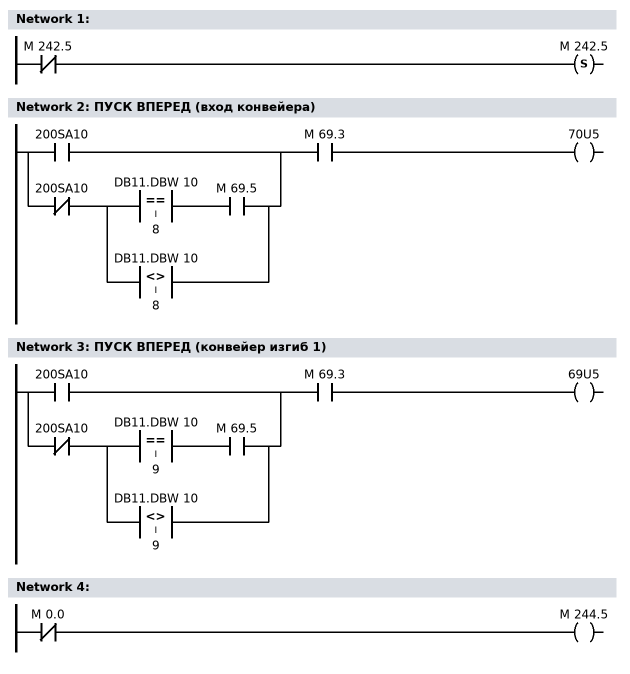
NETWORK
TITLE =
      AN    M 242.5;
      S     M 242.5;
NETWORK
TITLE = ПУСК ВПЕРЕД (вход конвейера)
      A(;
      O     "200SA10";
      O;
      AN    "200SA10";
      A(;
      A(;
      L     DB11.DBW 10;
      L     8;
      ==I;
      );
      A     M 69.5;
      O(;
      L     DB11.DBW 10;
      L     8;
      <>I;
      );
      );
      );
      A     M 69.3;
      =     "70U5";
NETWORK
TITLE = ПУСК ВПЕРЕД (конвейер изгиб 1)
      A(;
      O     "200SA10";
      O;
      AN    "200SA10";
      A(;
      A(;
      L     DB11.DBW 10;
      L     9;
      ==I;
      );
      A     M 69.5;
      O(;
      L     DB11.DBW 10;
      L     9;
      <>I;
      );
      );
      );
      A     M 69.3;
      =     "69U5";
NETWORK
TITLE =
      AN    M 0.0;
      =     M 244.5;
END_FUNCTION

FUNCTION FC 100 : VOID
VERSION : 0.1
BEGIN
// (block stored without names or comments; labels and parameter names are numbered)
NETWORK
TITLE =
      A     M 255.1;
      O(;
      A     DB11.DBX 1.6;
      A(;
      L     DB11.DBW 8;
      L     DB11.DBW 4;
      ==I;
      );
      );
      JCN   M001;
      AN    M 255.0;
      JCN   M001;
      L     DB11.DBW 4;
      L     100;
      +I;
      T     LW 100;
      L     101;
      <I;
      JC    M001;
      L     LW 100;
      L     104;
      >I;
      JC    M001;
      L     LW 100;
      OPN   DB [LW 100];
      CALL  "BLKMOV" (
           SRCBLK                   := P#DBX 0.0 BYTE 210,
           RET_VAL                  := LW 50,
           DSTBLK                   := P#DB99.DBX 0.0 BYTE 210);
M001: NOP   0;
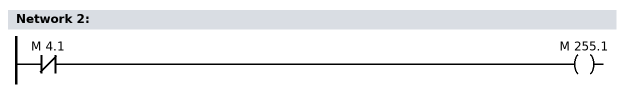
NETWORK
TITLE =
      AN    M 4.1;
      =     M 255.1;
NETWORK
TITLE =
      AN    DB11.DBX 2.0;
      JC    M002;
      L     DB11.DBW 8;
      L     100;
      +I;
      T     LW 100;
      L     101;
      <I;
      JC    M002;
      L     LW 100;
      L     104;
      >I;
      JC    M002;
      L     LW 100;
      OPN   DB [LW 100];
      CALL  "BLKMOV" (
           SRCBLK                   := P#DBX 0.0 BYTE 210,
           RET_VAL                  := LW 50,
           DSTBLK                   := P#DB100.DBX 0.0 BYTE 210);
      R     DB11.DBX 2.0;
M002: NOP   0;
NETWORK
TITLE =
      AN    DB11.DBX 1.6;
      JC    M003;
      L     DB11.DBW 8;
      L     100;
      +I;
      T     LW 100;
      L     101;
      <I;
      JC    M003;
      L     LW 100;
      L     104;
      >I;
      JC    M003;
      L     LW 100;
      OPN   DI [LW 100];
      CALL  "BLKMOV" (
           SRCBLK                   := P#DB100.DBX 0.0 BYTE 210,
           RET_VAL                  := LW 50,
           DSTBLK                   := P#DIX 0.0 BYTE 210);
      AN    T 1;
      JC    M003;
      R     DB11.DBX 1.6;
M003: NOP   0;
      A     DB11.DBX 1.6;
      L     S5T#1S;
      SD    T 1;
END_FUNCTION

FUNCTION FC 101 : VOID
VERSION : 0.1
BEGIN
// (block stored without names or comments; labels and parameter names are numbered)
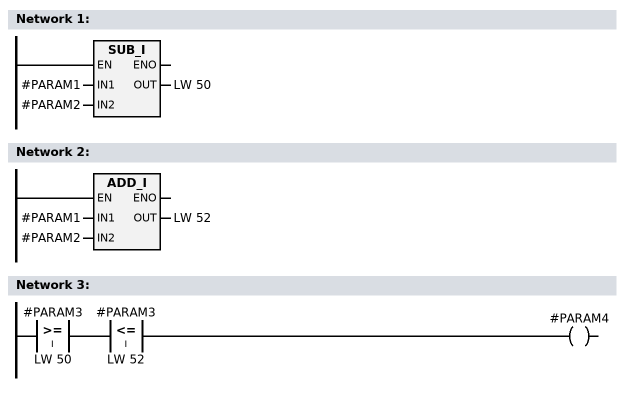
NETWORK
TITLE =
      L     #PARAM1;
      L     #PARAM2;
      -I;
      T     LW 50;
NETWORK
TITLE =
      L     #PARAM1;
      L     #PARAM2;
      +I;
      T     LW 52;
NETWORK
TITLE =
      A(;
      L     #PARAM3;
      L     LW 50;
      >=I;
      );
      A(;
      L     #PARAM3;
      L     LW 52;
      <=I;
      );
      =     #PARAM4;
END_FUNCTION

FUNCTION FC 102 : VOID
VERSION : 0.1
BEGIN
// (block stored without names or comments; labels and parameter names are numbered)
NETWORK
TITLE =
      L     DB12.DBW 516;
      L     256;
      >=I;
      JC    M001;
      L     DB12.DBW 516;
      L     2;
      *I;
      T     LD 0;
      L     LD 0;
      SLD   3;
      T     LD 0;
      L     DBW [LD 0];
      T     DB12.DBW 518;
      JU    M001;
      L     256;
      T     DB12.DBW 518;
M001: NOP   0;
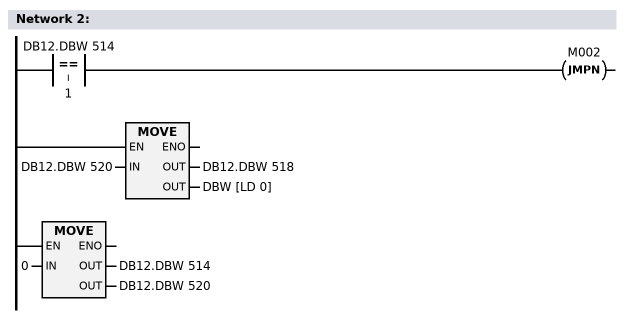
NETWORK
TITLE =
      L     DB12.DBW 514;
      L     1;
      ==I;
      JCN   M002;
      L     DB12.DBW 520;
      T     DB12.DBW 518;
      T     DBW [LD 0];
      L     0;
      T     DB12.DBW 514;
      T     DB12.DBW 520;
M002: NOP   0;
END_FUNCTION

FUNCTION FC 103 : VOID
VERSION : 0.1
BEGIN
// (block stored without names or comments; labels and parameter names are numbered)
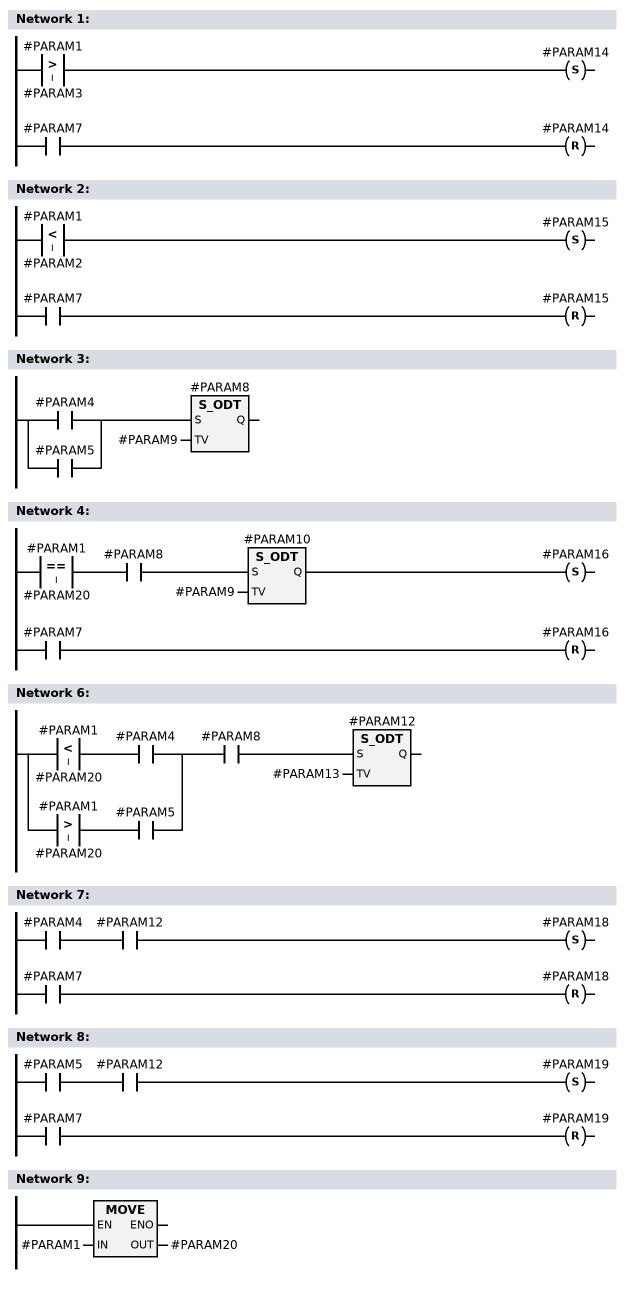
NETWORK
TITLE =
      A(;
      L     #PARAM1;
      L     #PARAM3;
      >I;
      );
      S     #PARAM14;
      A     #PARAM7;
      R     #PARAM14;
      NOP   0;
NETWORK
TITLE =
      A(;
      L     #PARAM1;
      L     #PARAM2;
      <I;
      );
      S     #PARAM15;
      A     #PARAM7;
      R     #PARAM15;
      NOP   0;
NETWORK
TITLE =
      A(;
      O     #PARAM4;
      O     #PARAM5;
      );
      L     #PARAM9;
      SD    #PARAM8;
      NOP   0;
      NOP   0;
      NOP   0;
      NOP   0;
NETWORK
TITLE =
      A(;
      A(;
      L     #PARAM1;
      L     #PARAM20;
      ==I;
      );
      A     #PARAM8;
      L     #PARAM9;
      SD    #PARAM10;
      NOP   0;
      NOP   0;
      NOP   0;
      A     #PARAM10;
      );
      S     #PARAM16;
      A     #PARAM7;
      R     #PARAM16;
      NOP   0;
NETWORK
TITLE =
      L     #PARAM20;
      L     #PARAM6;
      -I;
      T     LW 0;
      L     0;
      <I;
      JC    M001;
      JU    M002;
M001: L     0;
      T     LW 0;
M002: NOP   0;
      L     #PARAM20;
      L     #PARAM6;
      +I;
      T     LW 2;
      L     #PARAM1;
      L     LW 0;
      <I;
      JC    M003;
      L     #PARAM1;
      L     LW 2;
      >I;
      JC    M003;
      JU    M004;
M003: AN    #PARAM17;
      S     #PARAM17;
M004: R     #PARAM17;
NETWORK
TITLE =
      A(;
      A(;
      L     #PARAM1;
      L     #PARAM20;
      <I;
      );
      A     #PARAM4;
      O;
      A(;
      L     #PARAM1;
      L     #PARAM20;
      >I;
      );
      A     #PARAM5;
      );
      A     #PARAM8;
      L     #PARAM13;
      SD    #PARAM12;
      NOP   0;
      NOP   0;
      NOP   0;
      NOP   0;
NETWORK
TITLE =
      A     #PARAM4;
      A     #PARAM12;
      S     #PARAM18;
      A     #PARAM7;
      R     #PARAM18;
      NOP   0;
NETWORK
TITLE =
      A     #PARAM5;
      A     #PARAM12;
      S     #PARAM19;
      A     #PARAM7;
      R     #PARAM19;
      NOP   0;
NETWORK
TITLE =
      L     #PARAM1;
      T     #PARAM20;
END_FUNCTION

FUNCTION FC 104 : VOID
VERSION : 0.1
BEGIN
// (block stored without names or comments; labels and parameter names are numbered)
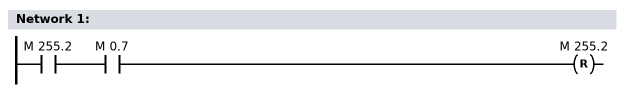
NETWORK
TITLE =
      A     M 255.2;
      A     M 0.7;
      R     M 255.2;
NETWORK
TITLE =
// (network holds code this reader does not know; not shown)
NETWORK
TITLE =
      L     MW 70;
      CAW;
      T     DB10.DBW 0;
      L     MW 72;
      CAW;
      T     DB10.DBW 2;
      L     MW 74;
      CAW;
      T     DB10.DBW 4;
      L     MW 76;
      CAW;
      T     DB10.DBW 6;
      L     MW 78;
      CAW;
      T     DB10.DBW 8;
      L     MW 80;
      CAW;
      T     DB10.DBW 10;
      L     MW 82;
      CAW;
      T     DB10.DBW 12;
      L     MW 84;
      CAW;
      T     DB10.DBW 14;
      L     MW 86;
      CAW;
      T     DB10.DBW 16;
      L     MW 88;
      CAW;
      T     DB10.DBW 18;
END_FUNCTION

FUNCTION FC 105 : VOID
VERSION : 0.1
BEGIN
// (block stored without names or comments; labels and parameter names are numbered)
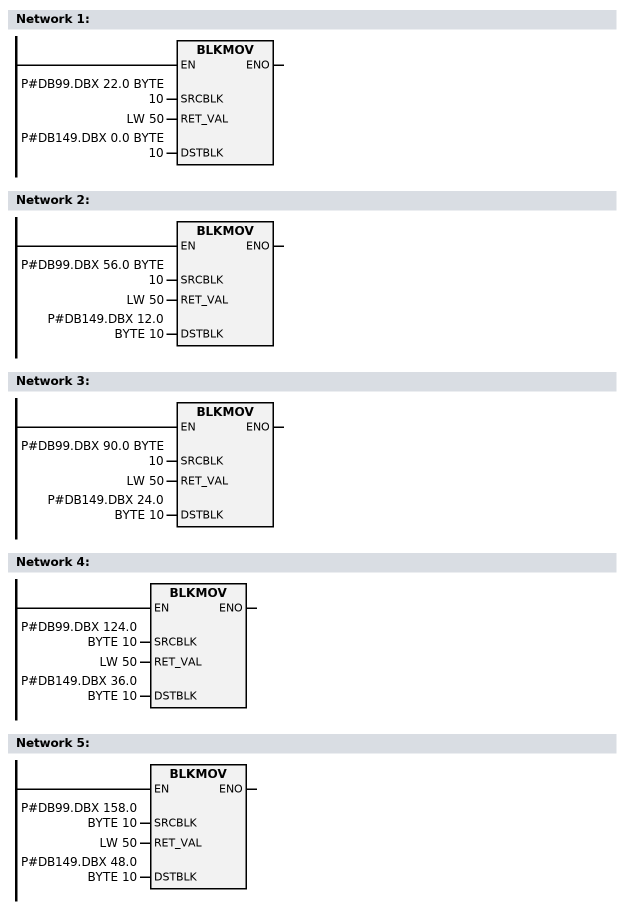
NETWORK
TITLE =
      CALL  "BLKMOV" (
           SRCBLK                   := P#DB99.DBX 22.0 BYTE 10,
           RET_VAL                  := LW 50,
           DSTBLK                   := P#DB149.DBX 0.0 BYTE 10);
NETWORK
TITLE =
      CALL  "BLKMOV" (
           SRCBLK                   := P#DB99.DBX 56.0 BYTE 10,
           RET_VAL                  := LW 50,
           DSTBLK                   := P#DB149.DBX 12.0 BYTE 10);
NETWORK
TITLE =
      CALL  "BLKMOV" (
           SRCBLK                   := P#DB99.DBX 90.0 BYTE 10,
           RET_VAL                  := LW 50,
           DSTBLK                   := P#DB149.DBX 24.0 BYTE 10);
NETWORK
TITLE =
      CALL  "BLKMOV" (
           SRCBLK                   := P#DB99.DBX 124.0 BYTE 10,
           RET_VAL                  := LW 50,
           DSTBLK                   := P#DB149.DBX 36.0 BYTE 10);
NETWORK
TITLE =
      CALL  "BLKMOV" (
           SRCBLK                   := P#DB99.DBX 158.0 BYTE 10,
           RET_VAL                  := LW 50,
           DSTBLK                   := P#DB149.DBX 48.0 BYTE 10);
END_FUNCTION

FUNCTION FC 110 : VOID
VERSION : 0.1
BEGIN
// (block stored without names or comments; labels and parameter names are numbered)
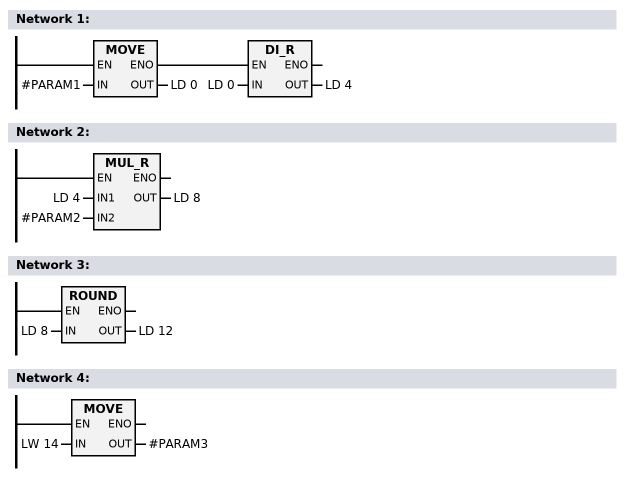
NETWORK
TITLE =
      A(;
      L     #PARAM1;
      T     LD 0;
      SET;
      SAVE;
      CLR;
      A     BR;
      );
      JNB   M001;
      L     LD 0;
      DTR;
      T     LD 4;
M001: NOP   0;
NETWORK
TITLE =
      L     LD 4;
      L     #PARAM2;
      *R;
      T     LD 8;
      NOP   0;
NETWORK
TITLE =
      L     LD 8;
      RND;
      T     LD 12;
      NOP   0;
NETWORK
TITLE =
      L     LW 14;
      T     #PARAM3;
      NOP   0;
END_FUNCTION

FUNCTION FC 111 : VOID
VERSION : 0.1
BEGIN
// (block stored without names or comments; labels and parameter names are numbered)
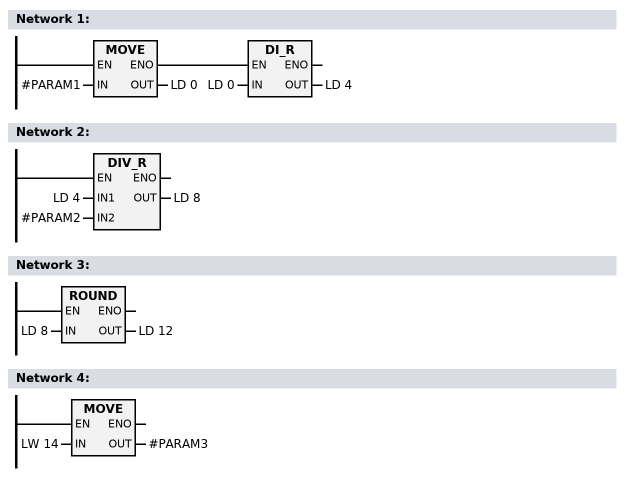
NETWORK
TITLE =
      A(;
      L     #PARAM1;
      T     LD 0;
      SET;
      SAVE;
      CLR;
      A     BR;
      );
      JNB   M001;
      L     LD 0;
      DTR;
      T     LD 4;
M001: NOP   0;
NETWORK
TITLE =
      L     LD 4;
      L     #PARAM2;
      /R;
      T     LD 8;
      NOP   0;
NETWORK
TITLE =
      L     LD 8;
      RND;
      T     LD 12;
      NOP   0;
NETWORK
TITLE =
      L     LW 14;
      T     #PARAM3;
      NOP   0;
END_FUNCTION

FUNCTION FC 112 : VOID
AUTHOR : sim
NAME : CTRL
VERSION : 1.0
BEGIN
// (block stored without names or comments; labels and parameter names are numbered)
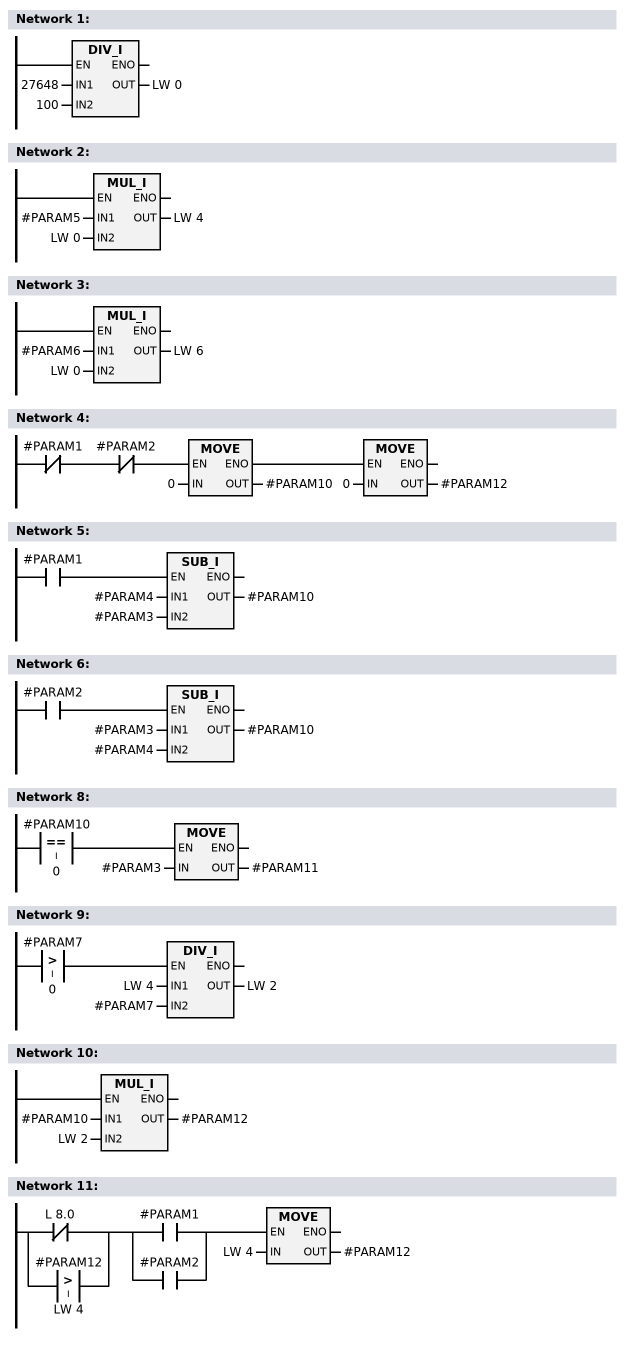
NETWORK
TITLE =
      L     27648;
      L     100;
      /I;
      T     LW 0;
      NOP   0;
NETWORK
TITLE =
      L     #PARAM5;
      L     LW 0;
      *I;
      T     LW 4;
      NOP   0;
NETWORK
TITLE =
      L     #PARAM6;
      L     LW 0;
      *I;
      T     LW 6;
      NOP   0;
NETWORK
TITLE =
      A(;
      AN    #PARAM1;
      AN    #PARAM2;
      JNB   M001;
      L     0;
      T     #PARAM10;
      SET;
      SAVE;
      CLR;
M001: A     BR;
      );
      JNB   M002;
      L     0;
      T     #PARAM12;
M002: NOP   0;
NETWORK
TITLE =
      A     #PARAM1;
      JNB   M003;
      L     #PARAM4;
      L     #PARAM3;
      -I;
      T     #PARAM10;
M003: NOP   0;
NETWORK
TITLE =
      A     #PARAM2;
      JNB   M004;
      L     #PARAM3;
      L     #PARAM4;
      -I;
      T     #PARAM10;
M004: NOP   0;
NETWORK
TITLE =
      A(;
      L     #PARAM10;
      L     0;
      <>I;
      );
      A(;
      L     #PARAM10;
      L     #PARAM7;
      <=I;
      );
      =     L 8.0;
NETWORK
TITLE =
      A(;
      L     #PARAM10;
      L     0;
      ==I;
      );
      JNB   M005;
      L     #PARAM3;
      T     #PARAM11;
M005: NOP   0;
NETWORK
TITLE =
      A(;
      L     #PARAM7;
      L     0;
      >I;
      );
      JNB   M006;
      L     LW 4;
      L     #PARAM7;
      /I;
      T     LW 2;
M006: NOP   0;
NETWORK
TITLE =
      L     #PARAM10;
      L     LW 2;
      *I;
      T     #PARAM12;
      NOP   0;
NETWORK
TITLE =
      A(;
      ON    L 8.0;
      O(;
      L     #PARAM12;
      L     LW 4;
      >I;
      );
      );
      A(;
      O     #PARAM1;
      O     #PARAM2;
      );
      JNB   M007;
      L     LW 4;
      T     #PARAM12;
M007: NOP   0;
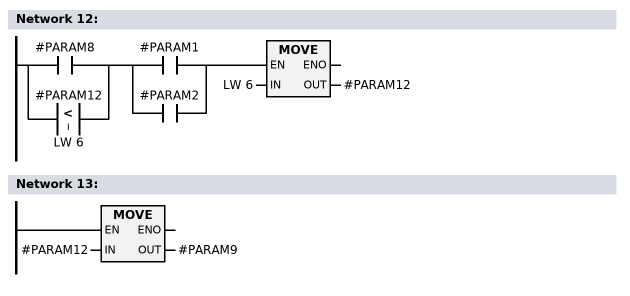
NETWORK
TITLE =
      A(;
      O     #PARAM8;
      O(;
      L     #PARAM12;
      L     LW 6;
      <I;
      );
      );
      A(;
      O     #PARAM1;
      O     #PARAM2;
      );
      JNB   M008;
      L     LW 6;
      T     #PARAM12;
M008: NOP   0;
NETWORK
TITLE =
      L     #PARAM12;
      T     #PARAM9;
      NOP   0;
END_FUNCTION

FUNCTION FC 113 : VOID
VERSION : 0.1
BEGIN
// (block stored without names or comments; labels and parameter names are numbered)
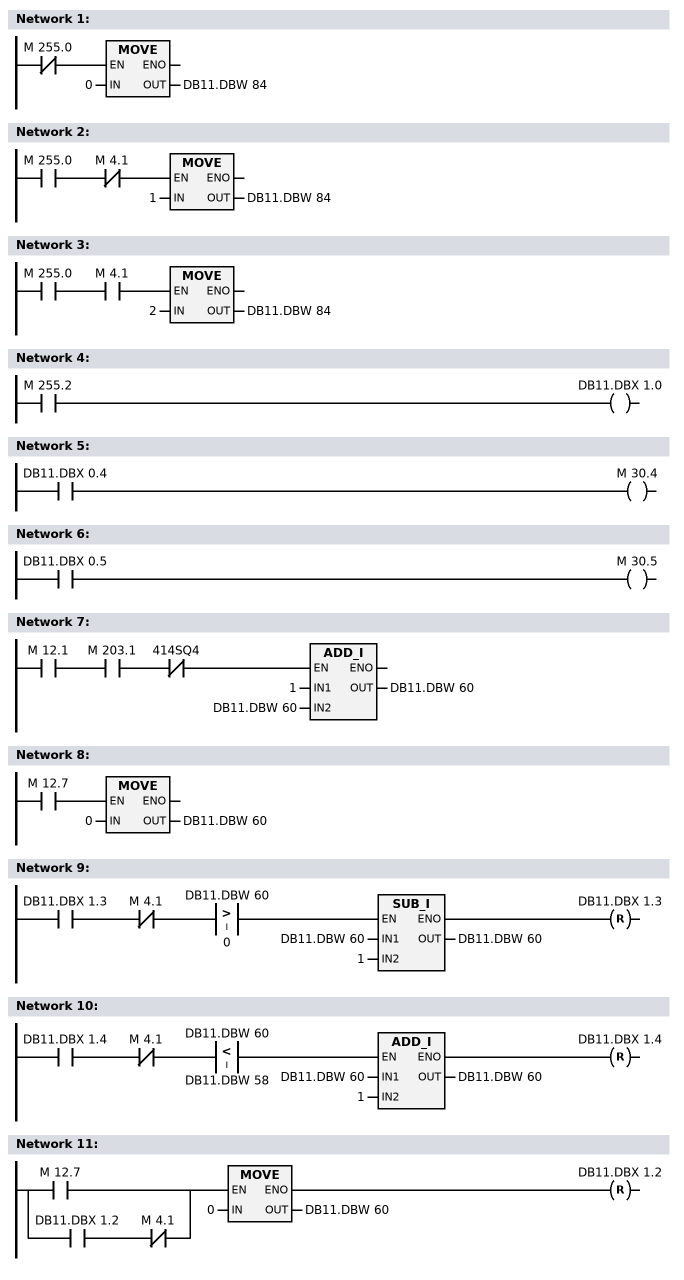
NETWORK
TITLE =
      AN    M 255.0;
      JNB   M001;
      L     0;
      T     DB11.DBW 84;
M001: NOP   0;
NETWORK
TITLE =
      A     M 255.0;
      AN    M 4.1;
      JNB   M002;
      L     1;
      T     DB11.DBW 84;
M002: NOP   0;
NETWORK
TITLE =
      A     M 255.0;
      A     M 4.1;
      JNB   M003;
      L     2;
      T     DB11.DBW 84;
M003: NOP   0;
NETWORK
TITLE =
      A     M 255.2;
      =     DB11.DBX 1.0;
NETWORK
TITLE =
      A     DB11.DBX 0.4;
      =     M 30.4;
NETWORK
TITLE =
      A     DB11.DBX 0.5;
      =     M 30.5;
NETWORK
TITLE =
      A     M 12.1;
      A     M 203.1;
      AN    "414SQ4";
      JNB   M004;
      L     1;
      L     DB11.DBW 60;
      +I;
      T     DB11.DBW 60;
M004: NOP   0;
NETWORK
TITLE =
      A     M 12.7;
      JNB   M005;
      L     0;
      T     DB11.DBW 60;
M005: NOP   0;
NETWORK
TITLE =
      A     DB11.DBX 1.3;
      AN    M 4.1;
      A(;
      L     DB11.DBW 60;
      L     0;
      >I;
      );
      JNB   M006;
      L     DB11.DBW 60;
      L     1;
      -I;
      T     DB11.DBW 60;
      AN    OV;
      SAVE;
      CLR;
M006: A     BR;
      R     DB11.DBX 1.3;
NETWORK
TITLE =
      A     DB11.DBX 1.4;
      AN    M 4.1;
      A(;
      L     DB11.DBW 60;
      L     DB11.DBW 58;
      <I;
      );
      JNB   M007;
      L     DB11.DBW 60;
      L     1;
      +I;
      T     DB11.DBW 60;
      AN    OV;
      SAVE;
      CLR;
M007: A     BR;
      R     DB11.DBX 1.4;
NETWORK
TITLE =
      A(;
      O     M 12.7;
      O;
      A     DB11.DBX 1.2;
      AN    M 4.1;
      );
      JNB   M008;
      L     0;
      T     DB11.DBW 60;
      SET;
      SAVE;
      CLR;
M008: A     BR;
      R     DB11.DBX 1.2;
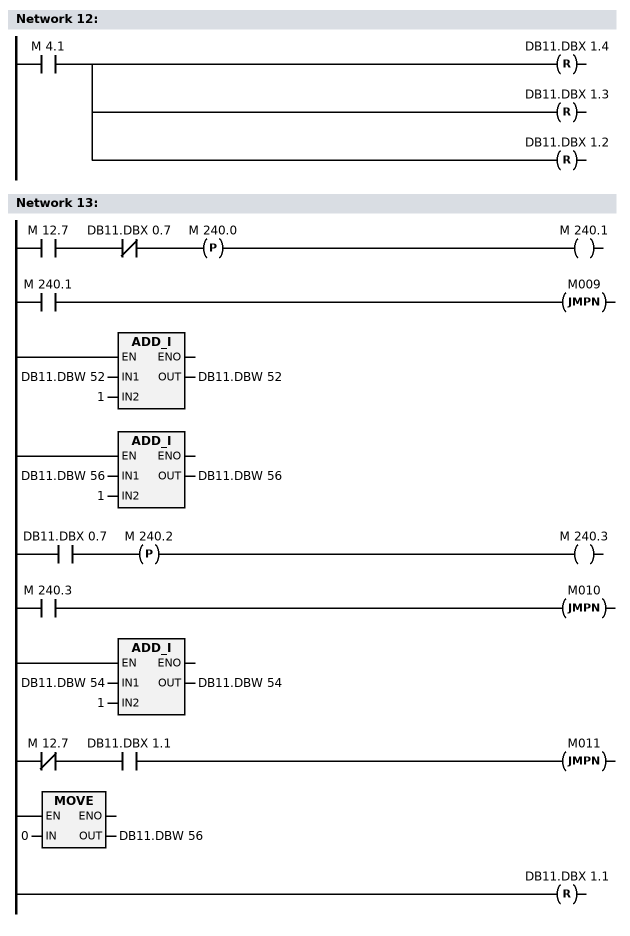
NETWORK
TITLE =
      A     M 4.1;
      R     DB11.DBX 1.4;
      R     DB11.DBX 1.3;
      R     DB11.DBX 1.2;
NETWORK
TITLE =
      A     M 12.7;
      AN    DB11.DBX 0.7;
      FP    M 240.0;
      =     M 240.1;
      A     M 240.1;
      JCN   M009;
      L     DB11.DBW 52;
      L     1;
      +I;
      T     DB11.DBW 52;
      L     DB11.DBW 56;
      L     1;
      +I;
      T     DB11.DBW 56;
M009: NOP   0;
      A     DB11.DBX 0.7;
      FP    M 240.2;
      =     M 240.3;
      A     M 240.3;
      JCN   M010;
      L     DB11.DBW 54;
      L     1;
      +I;
      T     DB11.DBW 54;
M010: NOP   0;
      AN    M 12.7;
      A     DB11.DBX 1.1;
      JCN   M011;
      L     0;
      T     DB11.DBW 56;
      R     DB11.DBX 1.1;
M011: NOP   0;
END_FUNCTION

// FC 125: know-how protected block, not included

FUNCTION FC 130 : VOID
AUTHOR : sim
NAME : CTRL
VERSION : 0.1
BEGIN
// (block stored without names or comments; labels and parameter names are numbered)
NETWORK
TITLE =
      A(;
      L     #PARAM1;
      L     #PARAM4;
      -I;
      L     #PARAM2;
      >I;
      );
      =     #PARAM7;
      R     #PARAM8;
NETWORK
TITLE =
      A(;
      L     #PARAM1;
      L     #PARAM3;
      +I;
      L     #PARAM2;
      <I;
      );
      =     #PARAM8;
      R     #PARAM7;
NETWORK
TITLE =
      AN    #PARAM7;
      AN    #PARAM8;
      =     #PARAM10;
NETWORK
TITLE =
      A     #PARAM7;
      A(;
      L     #PARAM1;
      L     #PARAM5;
      -I;
      L     #PARAM2;
      <=I;
      );
      =     L 0.0;
NETWORK
TITLE =
      A     #PARAM8;
      A(;
      L     #PARAM1;
      L     #PARAM6;
      +I;
      L     #PARAM2;
      >=I;
      );
      =     L 0.1;
NETWORK
TITLE =
      O     L 0.0;
      O     L 0.1;
      =     #PARAM9;
END_FUNCTION

FUNCTION FC 150 : VOID
VERSION : 0.1
BEGIN
// (block stored without names or comments; labels and parameter names are numbered)
NETWORK
TITLE =
      O(;
      L     #PARAM6;
      T     LW 0;
      SET;
      SAVE;
      CLR;
      A     BR;
      );
      O(;
      A     #PARAM2;
      JNB   M001;
      L     #PARAM7;
      T     LW 0;
      SET;
      SAVE;
      CLR;
M001: A     BR;
      );
      O(;
      A     #PARAM3;
      JNB   M002;
      L     #PARAM8;
      T     LW 0;
      SET;
      SAVE;
      CLR;
M002: A     BR;
      );
      O(;
      A     #PARAM4;
      JNB   M003;
      L     #PARAM9;
      T     LW 0;
      SET;
      SAVE;
      CLR;
M003: A     BR;
      );
      O(;
      A     #PARAM5;
      JNB   M004;
      L     #PARAM10;
      T     LW 0;
      SET;
      SAVE;
      CLR;
M004: A     BR;
      );
      =     L 2.0;
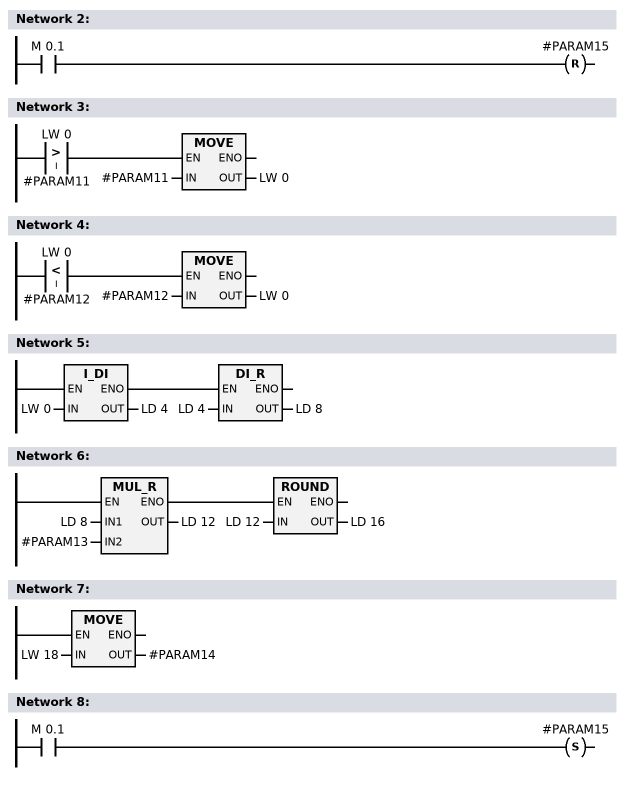
NETWORK
TITLE =
      A     M 0.1;
      R     #PARAM15;
NETWORK
TITLE =
      A(;
      L     LW 0;
      L     #PARAM11;
      >I;
      );
      JNB   M005;
      L     #PARAM11;
      T     LW 0;
M005: NOP   0;
NETWORK
TITLE =
      A(;
      L     LW 0;
      L     #PARAM12;
      <I;
      );
      JNB   M006;
      L     #PARAM12;
      T     LW 0;
M006: NOP   0;
NETWORK
TITLE =
      A(;
      L     LW 0;
      ITD;
      T     LD 4;
      SET;
      SAVE;
      CLR;
      A     BR;
      );
      JNB   M007;
      L     LD 4;
      DTR;
      T     LD 8;
M007: NOP   0;
NETWORK
TITLE =
      A(;
      L     LD 8;
      L     #PARAM13;
      *R;
      T     LD 12;
      AN    OV;
      SAVE;
      CLR;
      A     BR;
      );
      JNB   M008;
      L     LD 12;
      RND;
      T     LD 16;
M008: NOP   0;
NETWORK
TITLE =
      L     LW 18;
      T     #PARAM14;
      NOP   0;
NETWORK
TITLE =
      A     M 0.1;
      S     #PARAM15;
END_FUNCTION

FUNCTION FC 154 : VOID
AUTHOR : sim
NAME : DATA
VERSION : 0.1
BEGIN
// (block stored without names or comments; labels and parameter names are numbered)
NETWORK
TITLE =
      L     #PARAM1;
      T     LW 0;
      L     #PARAM3;
      T     LW 6;
      L     0;
      T     LW 12;
M001: L     LW 12;
      L     #PARAM5;
      <=I;
      JCN   M002;
      L     #PARAM2;
      L     LW 12;
      +I;
      L     2;
      *I;
      SLD   3;
      T     LD 2;
      L     #PARAM4;
      L     LW 12;
      +I;
      L     2;
      *I;
      SLD   3;
      T     LD 8;
      OPN   DB [LW 0];
      L     DBW [LD 2];
      OPN   DB [LW 6];
      T     DBW [LD 8];
      L     LW 12;
      L     1;
      +I;
      T     LW 12;
      JU    M001;
M002: NOP   0;
END_FUNCTION

FUNCTION FC 250 : VOID
//Вертикальное перемещение магнитной головы.
VERSION : 0.1
BEGIN
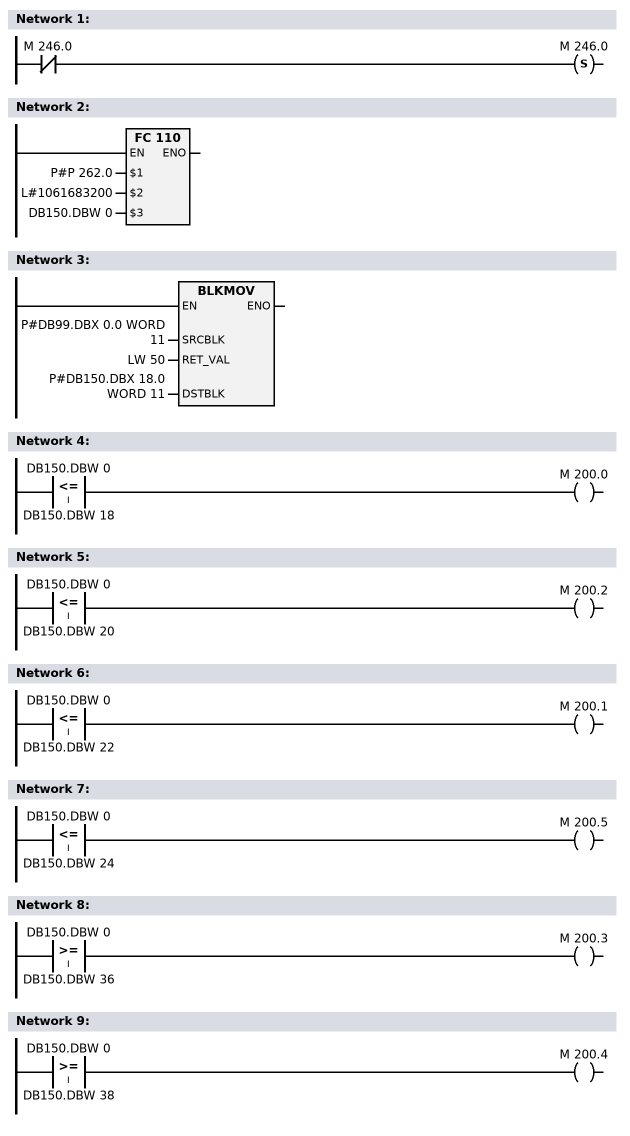
NETWORK
TITLE =
      AN    M 246.0;
      S     M 246.0;
NETWORK
TITLE =
      CALL  FC 110 (
           $1                       := P#P 262.0,
           $2                       := L#1061683200,
           $3                       := DB150.DBW 0);
NETWORK
TITLE =
      CALL  "BLKMOV" (
           SRCBLK                   := P#DB99.DBX 0.0 WORD 11,
           RET_VAL                  := LW 50,
           DSTBLK                   := P#DB150.DBX 18.0 WORD 11);
NETWORK
TITLE =
      L     DB150.DBW 0;
      L     DB150.DBW 18;
      <=I;
      =     M 200.0;
NETWORK
TITLE =
      L     DB150.DBW 0;
      L     DB150.DBW 20;
      <=I;
      =     M 200.2;
NETWORK
TITLE =
      L     DB150.DBW 0;
      L     DB150.DBW 22;
      <=I;
      =     M 200.1;
NETWORK
TITLE =
      L     DB150.DBW 0;
      L     DB150.DBW 24;
      <=I;
      =     M 200.5;
NETWORK
TITLE =
      L     DB150.DBW 0;
      L     DB150.DBW 36;
      >=I;
      =     M 200.3;
NETWORK
TITLE =
      L     DB150.DBW 0;
      L     DB150.DBW 38;
      >=I;
      =     M 200.4;
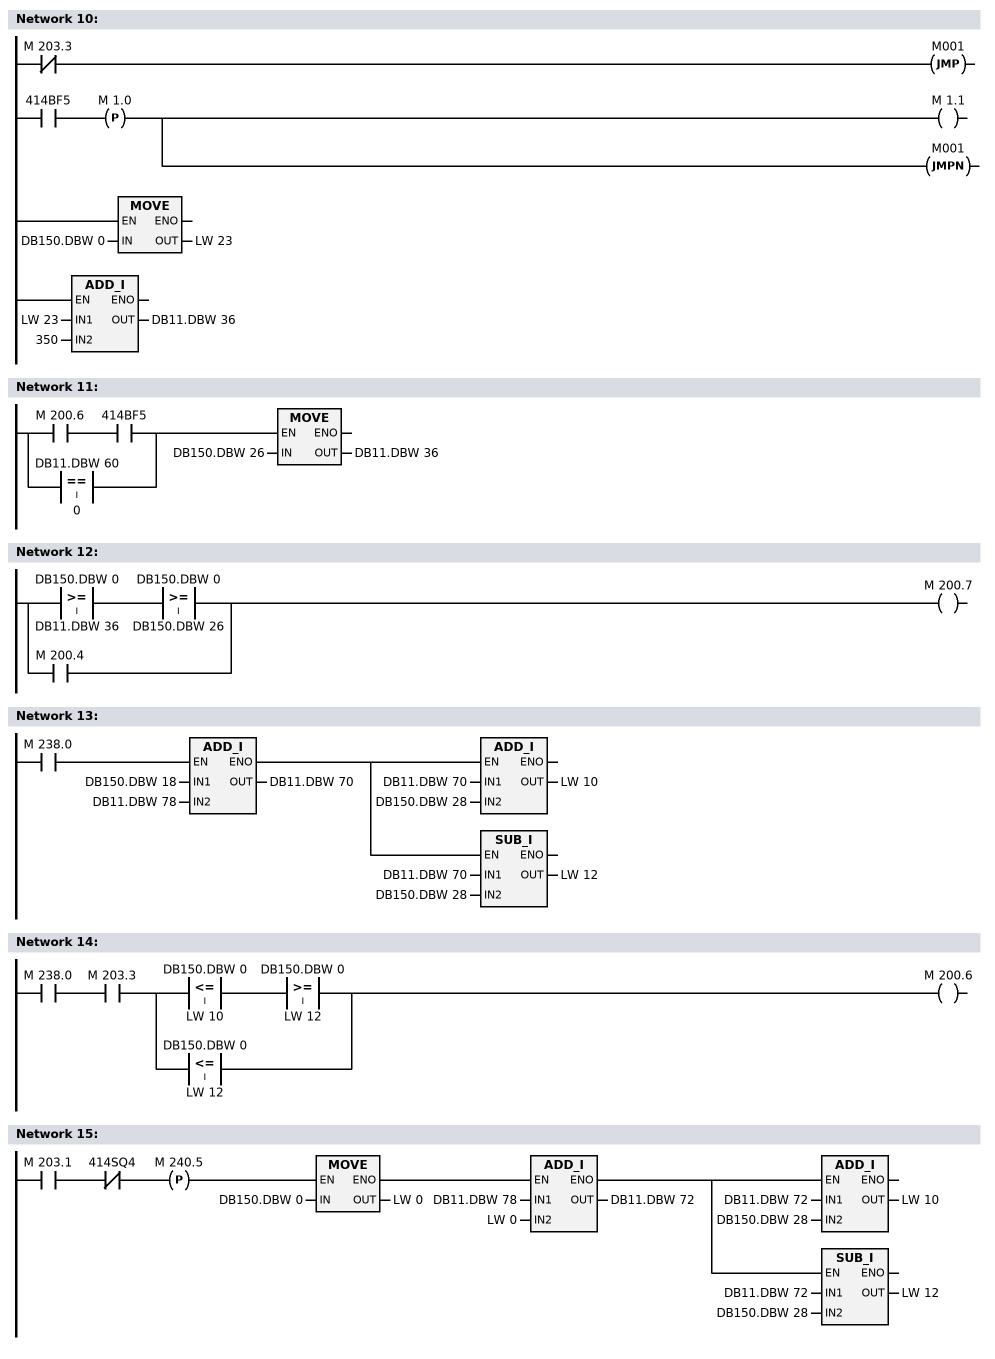
NETWORK
TITLE =
      AN    M 203.3;
      JC    M001;
      A     "414BF5";
      FP    M 1.0;
      =     M 1.1;
      JCN   M001;
      L     DB150.DBW 0;
      T     LW 23;
      L     LW 23;
      L     350;
      +I;
      T     DB11.DBW 36;
M001: NOP   0;
NETWORK
TITLE =
      A(;
      A     M 200.6;
      A     "414BF5";
      O(;
      L     DB11.DBW 60;
      L     0;
      ==I;
      );
      );
      JNB   _001;
      L     DB150.DBW 26;
      T     DB11.DBW 36;
_001: NOP   0;
NETWORK
TITLE =
      A(;
      L     DB150.DBW 0;
      L     DB11.DBW 36;
      >=I;
      );
      A(;
      L     DB150.DBW 0;
      L     DB150.DBW 26;
      >=I;
      );
      O     M 200.4;
      =     M 200.7;
NETWORK
TITLE =
      A     M 238.0;
      JNB   _002;
      L     DB150.DBW 18;
      L     DB11.DBW 78;
      +I;
      T     DB11.DBW 70;
      AN    OV;
      SAVE;
      CLR;
_002: A     BR;
      =     L 52.0;
      A     L 52.0;
      JNB   _007;
      L     DB11.DBW 70;
      L     DB150.DBW 28;
      +I;
      T     LW 10;
_007: NOP   0;
      A     L 52.0;
      JNB   _008;
      L     DB11.DBW 70;
      L     DB150.DBW 28;
      -I;
      T     LW 12;
_008: NOP   0;
NETWORK
TITLE =
      A     M 238.0;
      A     M 203.3;
      A(;
      A(;
      L     DB150.DBW 0;
      L     LW 10;
      <=I;
      );
      A(;
      L     DB150.DBW 0;
      L     LW 12;
      >=I;
      );
      O(;
      L     DB150.DBW 0;
      L     LW 12;
      <=I;
      );
      );
      =     M 200.6;
NETWORK
TITLE =
      A(;
      A     M 203.1;
      AN    "414SQ4";
      FP    M 240.5;
      JNB   _00e;
      L     DB150.DBW 0;
      T     LW 0;
      SET;
      SAVE;
      CLR;
_00e: A     BR;
      );
      JNB   _00f;
      L     DB11.DBW 78;
      L     LW 0;
      +I;
      T     DB11.DBW 72;
      AN    OV;
      SAVE;
      CLR;
_00f: A     BR;
      =     L 52.0;
      A     L 52.0;
      JNB   _010;
      L     DB11.DBW 72;
      L     DB150.DBW 28;
      +I;
      T     LW 10;
_010: NOP   0;
      A     L 52.0;
      JNB   _011;
      L     DB11.DBW 72;
      L     DB150.DBW 28;
      -I;
      T     LW 12;
_011: NOP   0;
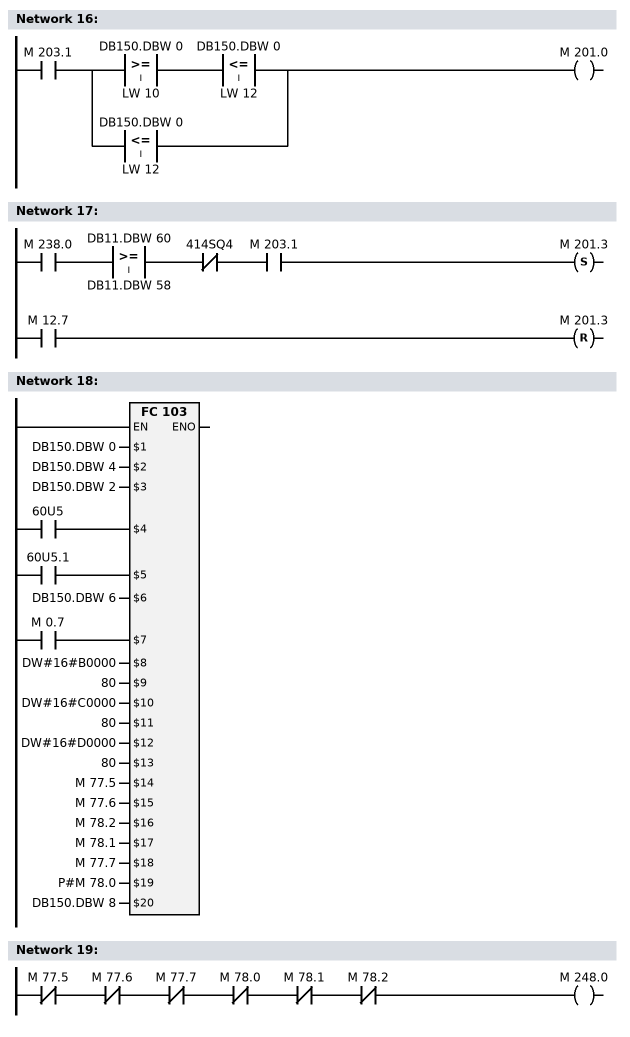
NETWORK
TITLE =
      A     M 203.1;
      A(;
      A(;
      L     DB150.DBW 0;
      L     LW 10;
      >=I;
      );
      A(;
      L     DB150.DBW 0;
      L     LW 12;
      <=I;
      );
      O(;
      L     DB150.DBW 0;
      L     LW 12;
      <=I;
      );
      );
      =     M 201.0;
NETWORK
TITLE =
      A     M 238.0;
      A(;
      L     DB11.DBW 60;
      L     DB11.DBW 58;
      >=I;
      );
      AN    "414SQ4";
      A     M 203.1;
      S     M 201.3;
      A     M 12.7;
      R     M 201.3;
      NOP   0;
NETWORK
TITLE =
      A     "60U5";
      =     L 52.0;
      BLD   103;
      A     "60U5.1";
      =     L 52.1;
      BLD   103;
      A     M 0.7;
      =     L 52.2;
      BLD   103;
      CALL  FC 103 (
           $1                       := DB150.DBW 0,
           $2                       := DB150.DBW 4,
           $3                       := DB150.DBW 2,
           $4                       := L 52.0,
           $5                       := L 52.1,
           $6                       := DB150.DBW 6,
           $7                       := L 52.2,
           $8                       := DW#16#B0000,
           $9                       := 80,
           $10                      := DW#16#C0000,
           $11                      := 80,
           $12                      := DW#16#D0000,
           $13                      := 80,
           $14                      := M 77.5,
           $15                      := M 77.6,
           $16                      := M 78.2,
           $17                      := M 78.1,
           $18                      := M 77.7,
           $19                      := P#M 78.0,
           $20                      := DB150.DBW 8);
      NOP   0;
NETWORK
TITLE =
      AN    M 77.5;
      AN    M 77.6;
      AN    M 77.7;
      AN    M 78.0;
      AN    M 78.1;
      AN    M 78.2;
      =     M 248.0;
END_FUNCTION

FUNCTION FC 251 : VOID
//Горизонтальное перемещение магнитной головы.
VERSION : 0.1
BEGIN
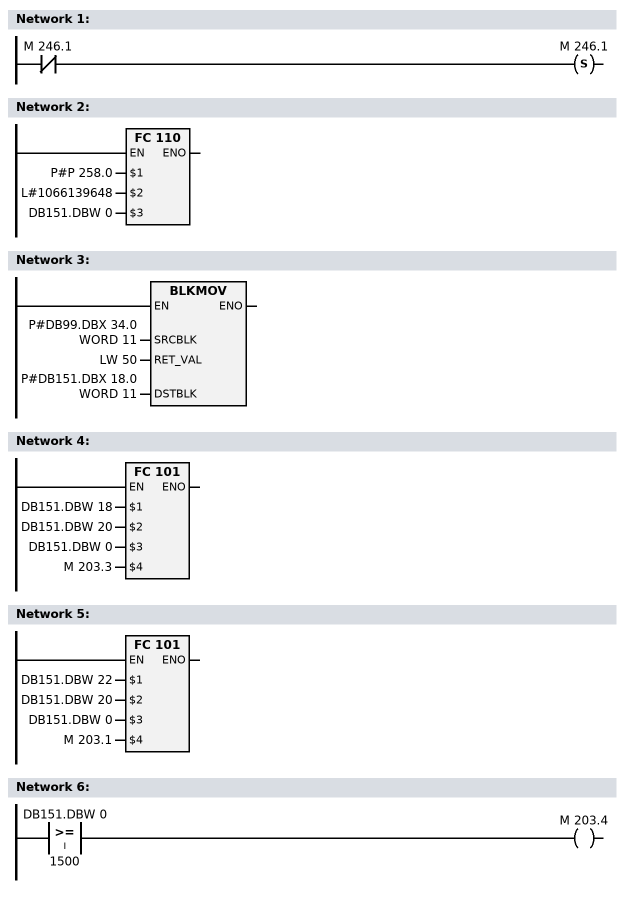
NETWORK
TITLE =
      AN    M 246.1;
      S     M 246.1;
NETWORK
TITLE =
      CALL  FC 110 (
           $1                       := P#P 258.0,
           $2                       := L#1066139648,
           $3                       := DB151.DBW 0);
NETWORK
TITLE =
      CALL  "BLKMOV" (
           SRCBLK                   := P#DB99.DBX 34.0 WORD 11,
           RET_VAL                  := LW 50,
           DSTBLK                   := P#DB151.DBX 18.0 WORD 11);
NETWORK
TITLE =
      CALL  FC 101 (
           $1                       := DB151.DBW 18,
           $2                       := DB151.DBW 20,
           $3                       := DB151.DBW 0,
           $4                       := M 203.3);
      NOP   0;
NETWORK
TITLE =
      CALL  FC 101 (
           $1                       := DB151.DBW 22,
           $2                       := DB151.DBW 20,
           $3                       := DB151.DBW 0,
           $4                       := M 203.1);
      NOP   0;
NETWORK
TITLE =
      L     DB151.DBW 0;
      L     1500;
      >=I;
      =     M 203.4;
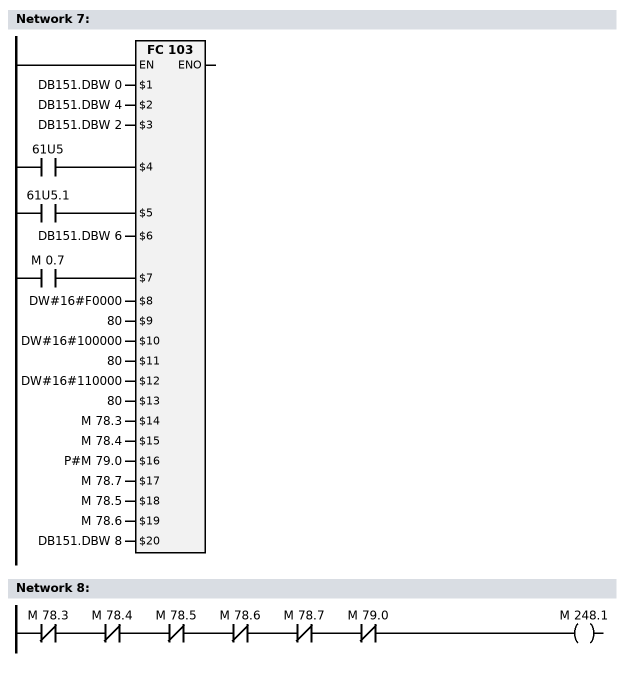
NETWORK
TITLE =
      A     "61U5";
      =     L 52.0;
      BLD   103;
      A     "61U5.1";
      =     L 52.1;
      BLD   103;
      A     M 0.7;
      =     L 52.2;
      BLD   103;
      CALL  FC 103 (
           $1                       := DB151.DBW 0,
           $2                       := DB151.DBW 4,
           $3                       := DB151.DBW 2,
           $4                       := L 52.0,
           $5                       := L 52.1,
           $6                       := DB151.DBW 6,
           $7                       := L 52.2,
           $8                       := DW#16#F0000,
           $9                       := 80,
           $10                      := DW#16#100000,
           $11                      := 80,
           $12                      := DW#16#110000,
           $13                      := 80,
           $14                      := M 78.3,
           $15                      := M 78.4,
           $16                      := P#M 79.0,
           $17                      := M 78.7,
           $18                      := M 78.5,
           $19                      := M 78.6,
           $20                      := DB151.DBW 8);
      NOP   0;
NETWORK
TITLE =
      AN    M 78.3;
      AN    M 78.4;
      AN    M 78.5;
      AN    M 78.6;
      AN    M 78.7;
      AN    M 79.0;
      =     M 248.1;
END_FUNCTION

FUNCTION FC 252 : VOID
//Вертикальное перемещение устройства размещения прокладок.
VERSION : 0.1
BEGIN
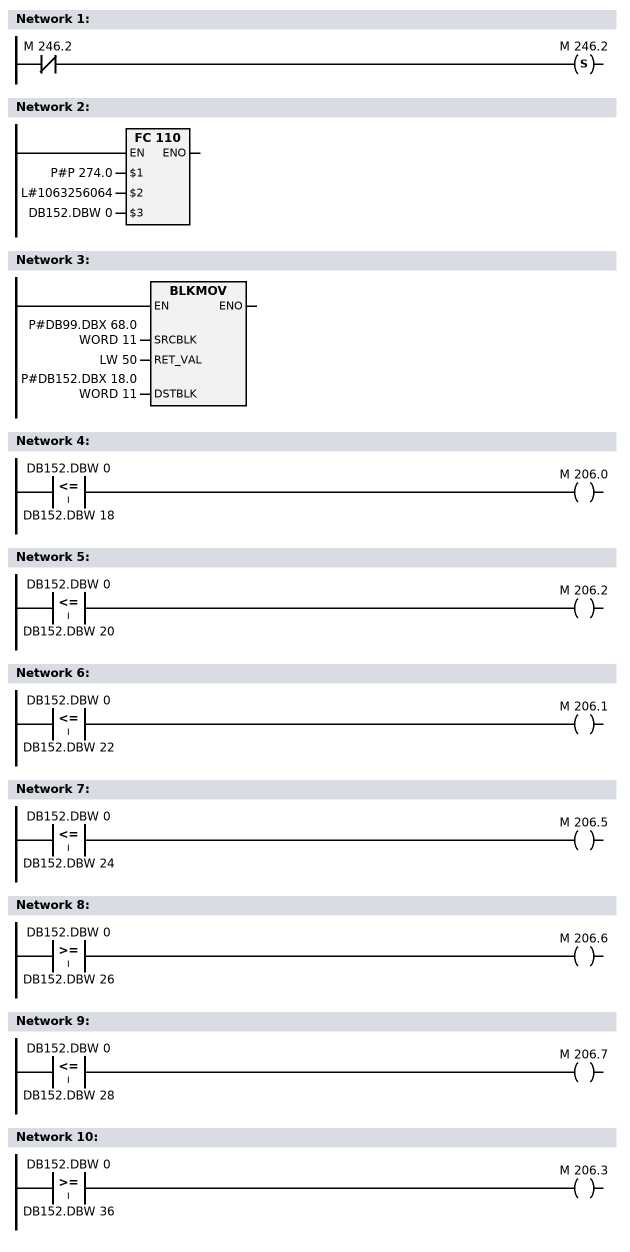
NETWORK
TITLE =
      AN    M 246.2;
      S     M 246.2;
NETWORK
TITLE =
      CALL  FC 110 (
           $1                       := P#P 274.0,
           $2                       := L#1063256064,
           $3                       := DB152.DBW 0);
NETWORK
TITLE =
      CALL  "BLKMOV" (
           SRCBLK                   := P#DB99.DBX 68.0 WORD 11,
           RET_VAL                  := LW 50,
           DSTBLK                   := P#DB152.DBX 18.0 WORD 11);
NETWORK
TITLE =
      L     DB152.DBW 0;
      L     DB152.DBW 18;
      <=I;
      =     M 206.0;
NETWORK
TITLE =
      L     DB152.DBW 0;
      L     DB152.DBW 20;
      <=I;
      =     M 206.2;
NETWORK
TITLE =
      L     DB152.DBW 0;
      L     DB152.DBW 22;
      <=I;
      =     M 206.1;
NETWORK
TITLE =
      L     DB152.DBW 0;
      L     DB152.DBW 24;
      <=I;
      =     M 206.5;
NETWORK
TITLE =
      L     DB152.DBW 0;
      L     DB152.DBW 26;
      >=I;
      =     M 206.6;
NETWORK
TITLE =
      L     DB152.DBW 0;
      L     DB152.DBW 28;
      <=I;
      =     M 206.7;
NETWORK
TITLE =
      L     DB152.DBW 0;
      L     DB152.DBW 36;
      >=I;
      =     M 206.3;
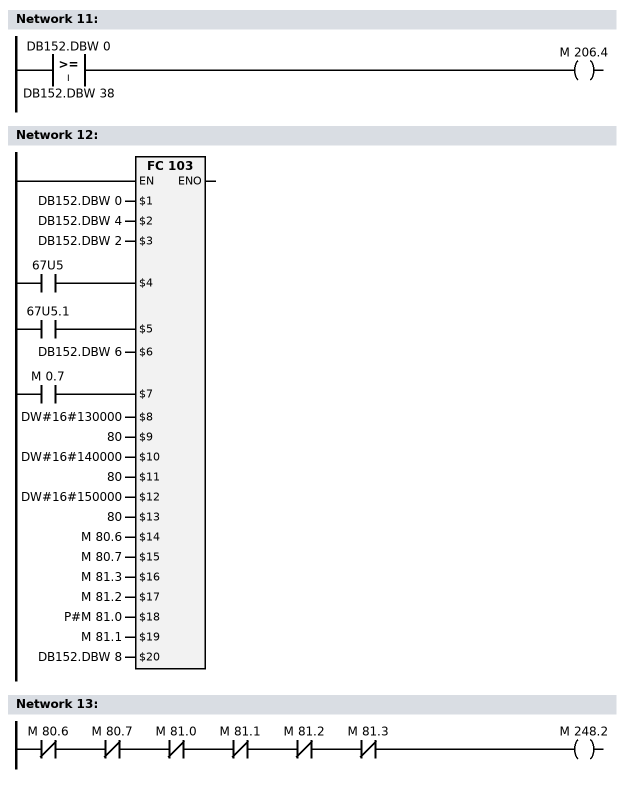
NETWORK
TITLE =
      L     DB152.DBW 0;
      L     DB152.DBW 38;
      >=I;
      =     M 206.4;
NETWORK
TITLE =
      A     "67U5";
      =     L 52.0;
      BLD   103;
      A     "67U5.1";
      =     L 52.1;
      BLD   103;
      A     M 0.7;
      =     L 52.2;
      BLD   103;
      CALL  FC 103 (
           $1                       := DB152.DBW 0,
           $2                       := DB152.DBW 4,
           $3                       := DB152.DBW 2,
           $4                       := L 52.0,
           $5                       := L 52.1,
           $6                       := DB152.DBW 6,
           $7                       := L 52.2,
           $8                       := DW#16#130000,
           $9                       := 80,
           $10                      := DW#16#140000,
           $11                      := 80,
           $12                      := DW#16#150000,
           $13                      := 80,
           $14                      := M 80.6,
           $15                      := M 80.7,
           $16                      := M 81.3,
           $17                      := M 81.2,
           $18                      := P#M 81.0,
           $19                      := M 81.1,
           $20                      := DB152.DBW 8);
      NOP   0;
NETWORK
TITLE =
      AN    M 80.6;
      AN    M 80.7;
      AN    M 81.0;
      AN    M 81.1;
      AN    M 81.2;
      AN    M 81.3;
      =     M 248.2;
END_FUNCTION

FUNCTION FC 253 : VOID
//Горизонтальное перемещение устройства размещения прокладок.
VERSION : 0.1
BEGIN
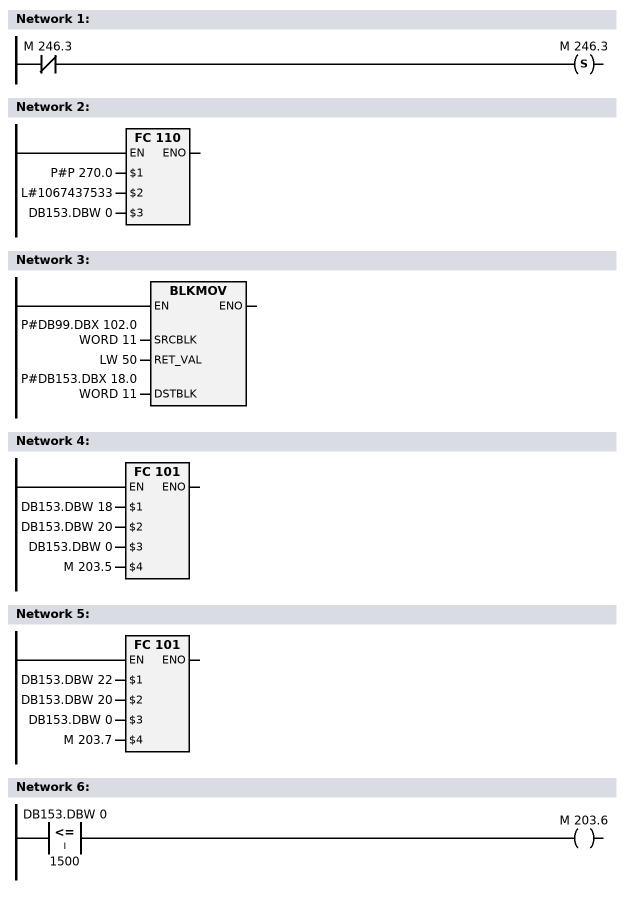
NETWORK
TITLE =
      AN    M 246.3;
      S     M 246.3;
NETWORK
TITLE =
      CALL  FC 110 (
           $1                       := P#P 270.0,
           $2                       := L#1067437533,
           $3                       := DB153.DBW 0);
NETWORK
TITLE =
      CALL  "BLKMOV" (
           SRCBLK                   := P#DB99.DBX 102.0 WORD 11,
           RET_VAL                  := LW 50,
           DSTBLK                   := P#DB153.DBX 18.0 WORD 11);
NETWORK
TITLE =
      CALL  FC 101 (
           $1                       := DB153.DBW 18,
           $2                       := DB153.DBW 20,
           $3                       := DB153.DBW 0,
           $4                       := M 203.5);
      NOP   0;
NETWORK
TITLE =
      CALL  FC 101 (
           $1                       := DB153.DBW 22,
           $2                       := DB153.DBW 20,
           $3                       := DB153.DBW 0,
           $4                       := M 203.7);
      NOP   0;
NETWORK
TITLE =
      L     DB153.DBW 0;
      L     1500;
      <=I;
      =     M 203.6;
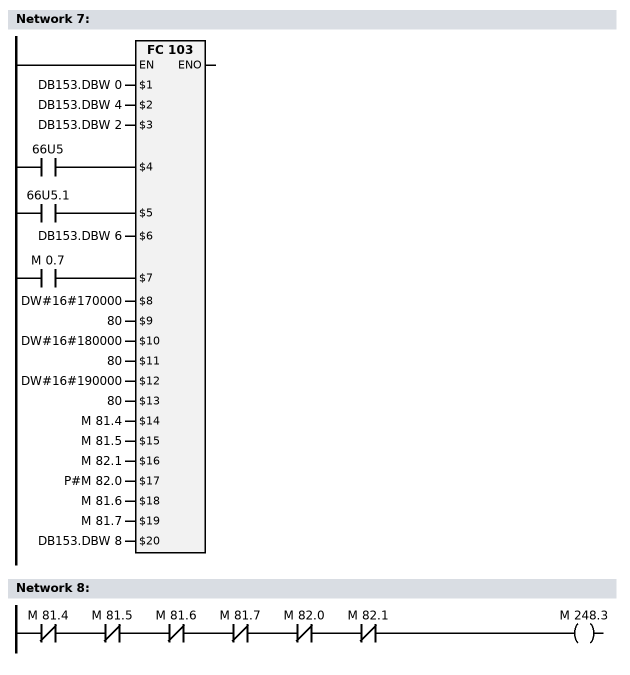
NETWORK
TITLE =
      A     "66U5";
      =     L 52.0;
      BLD   103;
      A     "66U5.1";
      =     L 52.1;
      BLD   103;
      A     M 0.7;
      =     L 52.2;
      BLD   103;
      CALL  FC 103 (
           $1                       := DB153.DBW 0,
           $2                       := DB153.DBW 4,
           $3                       := DB153.DBW 2,
           $4                       := L 52.0,
           $5                       := L 52.1,
           $6                       := DB153.DBW 6,
           $7                       := L 52.2,
           $8                       := DW#16#170000,
           $9                       := 80,
           $10                      := DW#16#180000,
           $11                      := 80,
           $12                      := DW#16#190000,
           $13                      := 80,
           $14                      := M 81.4,
           $15                      := M 81.5,
           $16                      := M 82.1,
           $17                      := P#M 82.0,
           $18                      := M 81.6,
           $19                      := M 81.7,
           $20                      := DB153.DBW 8);
      NOP   0;
NETWORK
TITLE =
      AN    M 81.4;
      AN    M 81.5;
      AN    M 81.6;
      AN    M 81.7;
      AN    M 82.0;
      AN    M 82.1;
      =     M 248.3;
END_FUNCTION

FUNCTION FC 254 : VOID
VERSION : 0.1
BEGIN
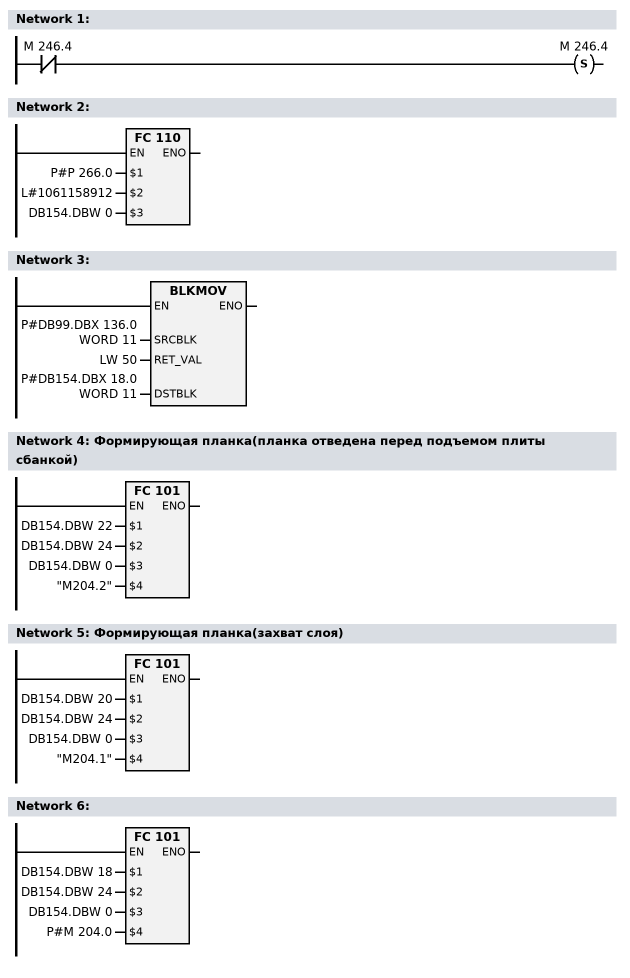
NETWORK
TITLE =
      AN    M 246.4;
      S     M 246.4;
NETWORK
TITLE =
      CALL  FC 110 (
           $1                       := P#P 266.0,
           $2                       := L#1061158912,
           $3                       := DB154.DBW 0);
NETWORK
TITLE =
      CALL  "BLKMOV" (
           SRCBLK                   := P#DB99.DBX 136.0 WORD 11,
           RET_VAL                  := LW 50,
           DSTBLK                   := P#DB154.DBX 18.0 WORD 11);
NETWORK
TITLE = Формирующая планка(планка отведена перед подъемом плиты сбанкой)
//М204.2 срабатывает когда In2 будет равен IN0. Уставка DB154.DBW22 должна быть 
//больше уставки DB154.DBW20 на 10-20 мм.
      CALL  FC 101 (
           $1                       := DB154.DBW 22,
           $2                       := DB154.DBW 24,
           $3                       := DB154.DBW 0,
           $4                       := "М204.2");
      NOP   0;
NETWORK
TITLE = Формирующая планка(захват слоя)
      CALL  FC 101 (
           $1                       := DB154.DBW 20,
           $2                       := DB154.DBW 24,
           $3                       := DB154.DBW 0,
           $4                       := "М204.1");
      NOP   0;
NETWORK
TITLE =
      CALL  FC 101 (
           $1                       := DB154.DBW 18,
           $2                       := DB154.DBW 24,
           $3                       := DB154.DBW 0,
           $4                       := P#M 204.0);
      NOP   0;
